{attribute 'GeneratedUsingTerminal: EJ2502-0000-0023'}
{attribute addProperty BoxType "EJ2502-0000-0023"}
{attribute addProperty Id "EtcSlaveTerminalBasePWM_Outputs_Channel_1AT %Q*PWM_Outputs_Channel_4C6289CD2PWM_Outputs_Channel_2AT %Q*PWM_Outputs_Channel_4C6289CD2WcStateAT %I*WcState_0B2B16F91InfoDataAT %I*InfoData_32EB74EA10"}
{attribute addProperty CRC "4287845392"}
{attribute addProperty Size "15"}
TYPE EJ2502_FF935410 EXTENDS EtcSlaveTerminalBase :
STRUCT
	{attribute addProperty Name "PWM_Outputs_Channel_1"}
	PWM_Outputs_Channel_1 : PWM_Outputs_Channel_4C6289CD;
	{attribute addProperty Name "PWM_Outputs_Channel_2"}
	PWM_Outputs_Channel_2 : PWM_Outputs_Channel_4C6289CD;
	{attribute addProperty Name "WcState"}
	WcState : WcState_0B2B16F9;
	{attribute addProperty Name "InfoData"}
	InfoData : InfoData_32EB74EA;
END_STRUCT
END_TYPE

(* stored: Version 1.2.0.0, ProductVersion 3.1.4024.9
   DUT EJ2502_FF935410: Id {338d8e6f-26f5-419a-8c39-7ce9e791f82c} *)
